{attribute 'qualified_only'}
VAR_GLOBAL
	On_DelayLED		:	TON;
	Off_DelayLED	:	TOF;
END_VAR

(* stored: Version 1.1.0.1, ProductVersion 3.1.4024.9
   GVL LEDTimer: Id {71533ef3-5567-44d6-ac89-352bfb3b71c3} *)
